TYPE U_SAFETY_RS :
UNION
	stStatusWords					: ST_SAFETY_FBStatus;			(* BUnknown, BState, wDiagnosis, wInputs, wOutputs - takie same dla wszystkich FB *)
	stStatus						: ST_SAFETY_RS; 				(* Rozbite na Bity - inne dla kazdego bloku*)
END_UNION
END_TYPE

(* stored: Version 1.1.0.1, ProductVersion 3.1.4022.12
   DUT U_SAFETY_RS: Id {709cb368-3305-4957-89a7-73ea2fd7881e} *)
